PROGRAM LampControl
VAR
END_VAR

GVL_General.fbMarqueeExPause();

//==========call the "Blinking" method ================================
//GVL_General.fbMarqueeExPause.Blinking(bStart:=GVL_Machine.HWIO.HWInput.StartBtn OR GVL_General.bStartBtnUI );

GVL_General.fbMarqueeExPause.Blinking(bStart:=GVL_SignalHanlding.fbHandleStartBtn.bSignalOutput OR GVL_General.bStartBtnUI );

END_PROGRAM

(* stored: Version 1.1.0.1, ProductVersion 3.1.4022.16
   POU LampControl: Id {3534f894-9fbd-456b-ae83-2812a303eb30}, SpecialFunc None *)
